{attribute 'qualified_only'}
{attribute 'strict'}
TYPE eTcoDataFormat :
(
	LittleEndian := 1,
	BigEndian := 2
);
END_TYPE

(* stored: Version 1.1.0.1, ProductVersion 3.1.4024.11
   DUT eTcoDataFormat: Id {550c8fe6-3655-00b9-0f57-e72ce5295107} *)
